// The station's data folder is an absolute path the medium creates on its first
// request (the press uses C:\ProgramData\Fraktal\PressDemo\).
METHOD A_file_medium_creates_its_folder
TEST('A_file_medium_creates_its_folder');
_t4(IN := _s4 < 99, PT := TEST_TIMEOUT);
IF _t4.Q AND (_s4 < 99) THEN
    AssertTrue(Condition := FALSE, Message := CONCAT('timed out in step ', INT_TO_STRING(_s4)));
    _s4 := 99;
    TEST_FINISHED();
    RETURN;
END_IF
_f4.Cyclic();
CASE _s4 OF
    0:
        AssertTrue(Condition := _m4.Setup(Folder := GENERIC_FOLDER, Where := Tc2_System.PATH_GENERIC),
            Message := 'an absolute folder is accepted');
        _k4 := _m4.M_StartWrite(Key := _M_Key(Name := 'Folder'), pData := ADR(_docA),
            Size := SIZEOF(_docA));
        _s4 := 1;
    1:
        IF _m4.M_Poll(Ticket := _k4, Result := _r4) THEN
            AssertTrue(Condition := _r4.Ok, Message := 'the document is written into the folder');
            _k4 := _m4.M_StartRead(Key := _M_Key(Name := 'Folder'), pData := ADR(_buf),
                Size := SIZEOF(_buf));
            _s4 := 2;
        END_IF
    2:
        IF _m4.M_Poll(Ticket := _k4, Result := _r4) THEN
            AssertTrue(Condition := _r4.Found AND (_r4.Length = SIZEOF(_docA)),
                Message := 'and read back from it');
            _f4.M_Delete(Path := CONCAT(GENERIC_FOLDER, CONCAT(_M_Key(Name := 'Folder'), '.a')),
                Where := Tc2_System.PATH_GENERIC);
            _s4 := 3;
        END_IF
    3:
        IF NOT _f4.Busy THEN
            AssertFalse(Condition := _f4.Error, Message := 'the file was where the medium said');
            _s4 := 99;
            TEST_FINISHED();
        END_IF
    99:
        ;
ELSE
    _s4 := 99;
END_CASE
END_METHOD

// Regression (live acceptance 2026-10-06): with the newest copy in slot a and an
// older one in slot b, a fresh run returned nothing - the payload check compared
// slot a against slot b's header - and its next write then replaced slot a, the
// newest copy. A fresh medium must read slot a, and must write the next copy to b.
METHOD The_newest_copy_wins_in_either_slot
VAR
    key : STRING(80);
END_VAR
TEST('The_newest_copy_wins_in_either_slot');
_t5(IN := _s5 < 99, PT := TEST_TIMEOUT);
IF _t5.Q AND (_s5 < 99) THEN
    AssertTrue(Condition := FALSE, Message := CONCAT('timed out in step ', INT_TO_STRING(_s5)));
    _s5 := 99;
    TEST_FINISHED();
    RETURN;
END_IF
key := _M_Key(Name := 'Slots');
_f5.Cyclic();
CASE _s5 OF
    0:      // generation 1 -> a, 2 -> b, 3 -> a
        _m5.Setup(Folder := '', Where := Tc2_System.PATH_BOOTPATH);
        _k5 := _m5.M_StartWrite(Key := key, pData := ADR(_docA), Size := SIZEOF(_docA));
        _s5 := 1;
    1:
        IF _m5.M_Poll(Ticket := _k5, Result := _r5) THEN
            _k5 := _m5.M_StartWrite(Key := key, pData := ADR(_docB), Size := SIZEOF(_docB));
            _s5 := 2;
        END_IF
    2:
        IF _m5.M_Poll(Ticket := _k5, Result := _r5) THEN
            _k5 := _m5.M_StartWrite(Key := key, pData := ADR(_docA), Size := SIZEOF(_docA));
            _s5 := 3;
        END_IF
    3:
        IF _m5.M_Poll(Ticket := _k5, Result := _r5) THEN
            AssertTrue(Condition := _r5.Ok, Message := 'three copies written');
            _m6.Setup(Folder := '', Where := Tc2_System.PATH_BOOTPATH);
            MEMSET(destAddr := ADR(_buf), fillByte := 0, n := SIZEOF(_buf));
            _k5 := _m6.M_StartRead(Key := key, pData := ADR(_buf), Size := SIZEOF(_buf));
            _s5 := 4;
        END_IF
    4:      // a fresh run reads the newest copy, which is in slot a
        IF _m6.M_Poll(Ticket := _k5, Result := _r5) THEN
            AssertTrue(Condition := _r5.Ok AND _r5.Found AND NOT _r5.Lost,
                Message := 'a fresh run finds the newest copy in slot a');
            AssertEquals_UDINT(Expected := SIZEOF(_docA), Actual := _r5.Length,
                Message := 'generation 3, not the older copy in slot b');
            _k5 := _m6.M_StartWrite(Key := key, pData := ADR(_docB), Size := SIZEOF(_docB));
            _s5 := 5;
        END_IF
    5:
        IF _m6.M_Poll(Ticket := _k5, Result := _r5) THEN
            AssertTrue(Condition := _r5.Ok, Message := 'generation 4 is written');
            // It must have replaced slot b: remove b and slot a still holds generation 3.
            _f5.M_Delete(Path := CONCAT(key, '.b'), Where := Tc2_System.PATH_BOOTPATH);
            _s5 := 6;
        END_IF
    6:
        IF NOT _f5.Busy THEN
            _m7.Setup(Folder := '', Where := Tc2_System.PATH_BOOTPATH);
            _k5 := _m7.M_StartRead(Key := key, pData := ADR(_buf), Size := SIZEOF(_buf));
            _s5 := 7;
        END_IF
    7:
        IF _m7.M_Poll(Ticket := _k5, Result := _r5) THEN
            AssertTrue(Condition := _r5.Found, Message := 'slot a was not overwritten');
            AssertEquals_UDINT(Expected := SIZEOF(_docA), Actual := _r5.Length,
                Message := 'the next write went to the slot without the newest copy');
            _f5.M_Delete(Path := CONCAT(key, '.a'), Where := Tc2_System.PATH_BOOTPATH);
            _s5 := 8;
        END_IF
    8:
        IF NOT _f5.Busy THEN
            _s5 := 99;
            TEST_FINISHED();
        END_IF
    99:
        ;
ELSE
    _s5 := 99;
END_CASE
END_METHOD

END_FUNCTION_BLOCK

// ---- Fraktal_Tests/FB_LiveConfig_Tests.TcPOU
// Core §3.8b under test: a root's live configuration and its parameter sets on a
// persistence medium, through the surface a station uses - SetPersistMedium and
// SetConfigStore - and the real file service of the test runtime.
//
// A "restart" is a second root instance with the same identity over the same
// files. Each test uses per-run names and removes what it wrote.
FUNCTION_BLOCK FB_LiveConfig_Tests EXTENDS TcUnit.FB_TestSuite
VAR
    _tag     : STRING(24);
    _name    : STRING(80);
    _garbage : ARRAY[0..15] OF BYTE := [16(16#5A)];
    _report  : ST_ReleaseReport;
    _s1 : INT;
    _t1 : TON;
    _m1 : FB_FilePersistMedium;
    _m2 : FB_FilePersistMedium;
    _r1 : FB_LocalRecipeProvider;
    _r2 : FB_LocalRecipeProvider;
    _rec0a, _recAa, _recBa : ST_ProbeModelParCfg;
    _rec0b, _recAb, _recBb : ST_ProbeModelParCfg;
    _u1 : FB_ProbeModelUnit;
    _u2 : FB_ProbeModelUnit;
    _u3 : FB_ProbeModelUnit;
    _f1 : FB_ProbeFileOps;
    _n1 : INT;
    _s2 : INT;
    _t2 : TON;
    _m3  : FB_FilePersistMedium;
    _m3b : FB_FilePersistMedium;
    _st1 : FB_MediumConfigStore;
    _st2 : FB_MediumConfigStore;
    _st3 : FB_MediumConfigStore;
    _f2 : FB_ProbeFileOps;
    _s3 : INT;
    _t3 : TON;
    _m4 : FB_FilePersistMedium;
    _st4 : FB_MediumConfigStore;
    _r4 : FB_LocalRecipeProvider;
    _rec4 : ST_ProbeModelParCfg;
    _u4 : FB_ProbeModelUnit;
    _f3 : FB_ProbeFileOps;
END_VAR
VAR CONSTANT
    TEST_TIMEOUT : TIME := T#60S;
END_VAR

IF _tag = '' THEN
    _tag := ULINT_TO_STRING(Tc2_Utilities.F_GetSystemTime() MOD 1000000000000);
    _name := CONCAT('Live', _tag);
END_IF
Station_and_model_data_come_back_from_their_documents();
Parameter_sets_come_back_from_the_medium();
A_saved_set_is_pending_until_its_document_is_written();

// Start names the restore while the documents are being read back.
METHOD PRIVATE _M_Restoring : BOOL
VAR_IN_OUT
    Unit : FB_ProbeModelUnit;
END_VAR
VAR
    i : INT;
END_VAR
_M_Restoring := FALSE;
Unit.ReleaseReportStart(Report := _report);
FOR i := 1 TO MIN(_report.Count, PL_Fraktal.MAX_RELEASE_REASONS) DO
    IF _report.Reasons[i].Description = 'std.release.configRestoring' THEN
        _M_Restoring := TRUE;
    END_IF
END_FOR
END_METHOD

// The n-th file of this root's live documents: station, then models 1 and 2,
// each slot a then b.
METHOD PRIVATE _M_LiveFile : STRING(255)
VAR_INPUT
    Index : INT;
END_VAR
VAR
    doc : STRING(40);
END_VAR
CASE Index / 2 OF
    0: doc := '.station';
    1: doc := '.model1';
ELSE
    doc := '.model2';
END_CASE
IF (Index MOD 2) = 0 THEN
    _M_LiveFile := CONCAT(_name, CONCAT(doc, '.a'));
ELSE
    _M_LiveFile := CONCAT(_name, CONCAT(doc, '.b'));
END_IF
END_METHOD

METHOD Station_and_model_data_come_back_from_their_documents
TEST('Station_and_model_data_come_back_from_their_documents');
_t1(IN := _s1 < 99, PT := TEST_TIMEOUT);
IF _t1.Q AND (_s1 < 99) THEN
    AssertTrue(Condition := FALSE, Message := CONCAT('timed out in step ', INT_TO_STRING(_s1)));
    _s1 := 99;
    TEST_FINISHED();
    RETURN;
END_IF
_f1.Cyclic();
CASE _s1 OF
    0:      // first run
        _rec0a.Speed := 1;
        _recAa.Speed := 10;
        _recBa.Speed := 20;
        _r1.Register(ModelCode := '', RecipeKey := 'ProbeModel', pData := ADR(_rec0a), Size := SIZEOF(_rec0a));
        _r1.Register(ModelCode := 'A', RecipeKey := 'ProbeModel', pData := ADR(_recAa), Size := SIZEOF(_recAa));
        _r1.Register(ModelCode := 'B', RecipeKey := 'ProbeModel', pData := ADR(_recBa), Size := SIZEOF(_recBa));
        _u1.ParCfg := _rec0a;
        _u1.Setup(Name := _name, Provider := _r1);
        _m1.Setup(Folder := '', Where := Tc2_System.PATH_BOOTPATH);
        AssertTrue(Condition := _u1.SetPersistMedium(Medium := _m1), Message := 'the medium is accepted');
        _u1();
        AssertFalse(Condition := _u1.WriteConfig(TargetPath := _name, WriteKey := 'probe.limit',
            Revision := 1, TextValue := '42'),
            Message := 'a write before the documents are back is refused: the restore would replay over it');
        AssertTrue(Condition := _M_Restoring(Unit := _u1), Message := 'and Start names the restore');
        _s1 := 1;
    1:
        _u1();
        IF NOT _M_Restoring(Unit := _u1) THEN
            AssertFalse(Condition := _u1.ConfigPersist.RestoreLost,
                Message := 'documents that never existed lost nothing');
            AssertTrue(Condition := _u1.WriteConfig(TargetPath := _name, WriteKey := 'probe.limit',
                Revision := 1, TextValue := '42'), Message := 'a station value is written');
            AssertTrue(Condition := _u1.WriteModelConfig(ModelIndex := 2, TargetPath := _name,
                WriteKey := 'probe.speed', Revision := 1, TextValue := '25'),
                Message := 'a model value of model B is written');
            AssertTrue(Condition := _u1.ConfigPersist.Pending, Message := 'live, not yet durable');
            _s1 := 2;
        END_IF
    2:
        _u1();
        IF NOT _u1.ConfigPersist.Pending THEN
            AssertFalse(Condition := _u1.ConfigPersist.Failed,
                Message := 'the documents are written within the declared window');
            _s1 := 3;
        END_IF
    3:      // restart: a new instance of the same root over the same files
        _rec0b.Speed := 1;
        _recAb.Speed := 10;
        _recBb.Speed := 20;
        _r2.Register(ModelCode := '', RecipeKey := 'ProbeModel', pData := ADR(_rec0b), Size := SIZEOF(_rec0b));
        _r2.Register(ModelCode := 'A', RecipeKey := 'ProbeModel', pData := ADR(_recAb), Size := SIZEOF(_recAb));
        _r2.Register(ModelCode := 'B', RecipeKey := 'ProbeModel', pData := ADR(_recBb), Size := SIZEOF(_recBb));
        _u2.ParCfg := _rec0b;
        _u2.Setup(Name := _name, Provider := _r2);
        _m2.Setup(Folder := '', Where := Tc2_System.PATH_BOOTPATH);
        _u2.SetPersistMedium(Medium := _m2);
        _u2();
        _s1 := 4;
    4:
        _u2();
        IF NOT _M_Restoring(Unit := _u2) THEN
            AssertEquals_DINT(Expected := 42, Actual := _u2.StationLimit,
                Message := 'the station value comes back from its document');
            AssertEquals_DINT(Expected := 25, Actual := _recBb.Speed,
                Message := 'model B$'s value comes back into B$'s record');
            AssertEquals_DINT(Expected := 10, Actual := _recAb.Speed,
                Message := 'model A keeps its own value');
            AssertFalse(Condition := _u2.ConfigPersist.RestoreLost, Message := 'nothing was lost');
            _s1 := 5;
        END_IF
    5:      // damage both copies of the station document
        _u2();
        IF NOT _u2.ConfigPersist.Pending AND _f1.M_Write(Path := _M_LiveFile(Index := 0),
                Where := Tc2_System.PATH_BOOTPATH, pData := ADR(_garbage), Size := SIZEOF(_garbage)) THEN
            _s1 := 6;
        END_IF
    6:
        IF NOT _f1.Busy AND _f1.M_Write(Path := _M_LiveFile(Index := 1),
                Where := Tc2_System.PATH_BOOTPATH, pData := ADR(_garbage), Size := SIZEOF(_garbage)) THEN
            _s1 := 7;
        END_IF
    7:      // restart over the medium that confirmed the writes
        IF NOT _f1.Busy THEN
            _u3.ParCfg := _rec0b;
            _u3.Setup(Name := _name, Provider := _r2);
            _u3.SetPersistMedium(Medium := _m2);
            _u3();
            _s1 := 8;
        END_IF
    8:
        _u3();
        IF NOT _M_Restoring(Unit := _u3) THEN
            _u3();                      // the loss is drained on the next scan
            AssertTrue(Condition := _u3.ConfigPersist.RestoreLost,
                Message := 'a station document confirmed and then lost is a loss (3.8b)');
            AssertEquals_STRING(Expected := CONCAT(_name, '.station'),
                Actual := _u3.ConfigPersist.LostPath, Message := 'named by its document');
            AssertTrue(Condition := F_ProbeAlarmActive(pLog := ADR(_u3.AlarmLog),
                Reason := E_Reason.CONFIG_RESTORE_LOST, Source := CONCAT(_name, '.station')),
                Message := 'and announced');
            AssertEquals_DINT(Expected := 5, Actual := _u3.StationLimit,
                Message := 'nothing is taken from a damaged document');
            AssertEquals_DINT(Expected := 25, Actual := _recBb.Speed,
                Message := 'an intact model document still restores');
            _s1 := 9;
        END_IF
    9:      // the baseline is rewritten; then remove every file
        _u3();
        IF NOT _u3.ConfigPersist.Pending THEN
            _n1 := 0;
            _s1 := 10;
        END_IF
    10:
        IF _n1 > 5 THEN
            _s1 := 99;
            TEST_FINISHED();
        ELSIF NOT _f1.Busy AND _f1.M_Delete(Path := _M_LiveFile(Index := _n1),
                Where := Tc2_System.PATH_BOOTPATH) THEN
            _n1 := _n1 + 1;
        END_IF
    99:
        ;
ELSE
    _s1 := 99;
END_CASE
END_METHOD

METHOD Parameter_sets_come_back_from_the_medium
VAR
    info   : ST_ConfigSetInfo;
    record : ST_ConfigRecord;
    prefix : STRING(60);
END_VAR
TEST('Parameter_sets_come_back_from_the_medium');
_t2(IN := _s2 < 99, PT := TEST_TIMEOUT);
IF _t2.Q AND (_s2 < 99) THEN
    AssertTrue(Condition := FALSE, Message := CONCAT('timed out in step ', INT_TO_STRING(_s2)));
    _s2 := 99;
    TEST_FINISHED();
    RETURN;
END_IF
prefix := CONCAT('FrkSets_', _tag);
_f2.Cyclic();
CASE _s2 OF
    0:
        _m3.Setup(Folder := '', Where := Tc2_System.PATH_BOOTPATH);
        AssertTrue(Condition := _st1.Setup(Medium := _m3, KeyPrefix := prefix),
            Message := 'the store takes the medium');
        info.SetName := 'Recipe';
        info.RootIdentity := 'Test.Sets';
        info.SetSchema := 1;
        info.ConfigRev := 7;
        info.Kind := E_ConfigKind.STATION_CFG;
        AssertFalse(Condition := _st1.M_SaveBegin(Info := info),
            Message := 'no save before the stored sets are back');
        _s2 := 1;
    1:
        _st1.M_Cyclic();
        IF _st1.Restored THEN
            AssertEquals_INT(Expected := 0, Actual := _st1.M_Count(), Message := 'an empty medium');
            AssertFalse(Condition := _st1.RestoreLost, Message := 'lost nothing');
            info.SetName := 'Recipe';
            info.RootIdentity := 'Test.Sets';
            info.SetSchema := 1;
            info.ConfigRev := 7;
            info.Kind := E_ConfigKind.STATION_CFG;
            AssertTrue(Condition := _st1.M_SaveBegin(Info := info), Message := 'a save opens');
            record.Scope := 'Test.Sets';
            record.WriteKey := 'probe.limit';
            record.Revision := 1;
            record.Kind := E_ConfigKind.STATION_CFG;
            record.ValueType := E_ConfigValueType.NUMBER;
            record.ValueText := '42';
            _st1.M_SaveRecord(Record := record);
            record.WriteKey := 'probe.text';
            record.ValueType := E_ConfigValueType.TEXT;
            record.ValueText := 'with "quotes", a \ and a , comma';
            _st1.M_SaveRecord(Record := record);
            AssertTrue(Condition := _st1.M_SaveCommit(), Message := 'and commits');
            AssertFalse(Condition := _st1.Durable, Message := 'live, not yet written');
            _s2 := 2;
        END_IF
    2:
        _st1.M_Cyclic();
        IF _st1.Durable THEN
            _m3b.Setup(Folder := '', Where := Tc2_System.PATH_BOOTPATH);
            _st2.Setup(Medium := _m3b, KeyPrefix := prefix);
            _s2 := 3;
        END_IF
    3:
        _st2.M_Cyclic();
        IF _st2.Restored THEN
            AssertEquals_INT(Expected := 1, Actual := _st2.M_Count(), Message := 'the set comes back');
            AssertTrue(Condition := _st2.M_ReadInfo(SetName := 'Recipe', Info := info),
                Message := 'under its name');
            AssertEquals_INT(Expected := 2, Actual := info.RecordCount, Message := 'whole');
            AssertEquals_STRING(Expected := 'Test.Sets', Actual := info.RootIdentity,
                Message := 'with the identity of the root that took it');
            AssertTrue(Condition := _st2.M_ReadRecord(SetName := 'Recipe', Index := 2,
                Record := record), Message := 'a record reads back');
            AssertEquals_STRING(Expected := 'with "quotes", a \ and a , comma',
                Actual := record.ValueText, Message := 'a text value survives the file exactly');
            AssertTrue(Condition := _st2.M_Delete(SetName := 'Recipe'), Message := 'the set is deleted');
            _s2 := 4;
        END_IF
    4:
        _st2.M_Cyclic();
        IF _st2.Durable THEN
            _st3.Setup(Medium := _m3b, KeyPrefix := prefix);
            _s2 := 5;
        END_IF
    5:
        _st3.M_Cyclic();
        IF _st3.Restored THEN
            AssertEquals_INT(Expected := 0, Actual := _st3.M_Count(),
                Message := 'a deleted set stays deleted');
            AssertFalse(Condition := _st3.RestoreLost, Message := 'by intent, not lost');
            _f2.M_Delete(Path := CONCAT(prefix, '.set1.a'), Where := Tc2_System.PATH_BOOTPATH);
            _s2 := 6;
        END_IF
    6:
        IF NOT _f2.Busy THEN
            _f2.M_Delete(Path := CONCAT(prefix, '.set1.b'), Where := Tc2_System.PATH_BOOTPATH);
            _s2 := 7;
        END_IF
    7:
        IF NOT _f2.Busy THEN
            _s2 := 99;
            TEST_FINISHED();
        END_IF
    99:
        ;
ELSE
    _s2 := 99;
END_CASE
END_METHOD

// The root finds the store's own writer (__QUERYINTERFACE) and drives it, so a
// saved set is PersistPending until its document is written - one SetConfigStore.
METHOD A_saved_set_is_pending_until_its_document_is_written
VAR
    prefix : STRING(60);
END_VAR
TEST('A_saved_set_is_pending_until_its_document_is_written');
_t3(IN := _s3 < 99, PT := TEST_TIMEOUT);
IF _t3.Q AND (_s3 < 99) THEN
    AssertTrue(Condition := FALSE, Message := CONCAT('timed out in step ', INT_TO_STRING(_s3)));
    _s3 := 99;
    TEST_FINISHED();
    RETURN;
END_IF
prefix := CONCAT('FrkRootSets_', _tag);
_f3.Cyclic();
CASE _s3 OF
    0:
        _rec4.Speed := 3;
        _r4.Register(ModelCode := '', RecipeKey := 'ProbeModel', pData := ADR(_rec4), Size := SIZEOF(_rec4));
        _u4.ParCfg := _rec4;
        _u4.Setup(Name := CONCAT('Sets', _tag), Provider := _r4);
        _m4.Setup(Folder := '', Where := Tc2_System.PATH_BOOTPATH);
        _st4.Setup(Medium := _m4, KeyPrefix := prefix);
        AssertTrue(Condition := _u4.SetConfigStore(Store := _st4), Message := 'the store is wired');
        _u4();
        _s3 := 1;
    1:
        _u4();                          // the root, not the test, drives the store
        IF _st4.Restored THEN
            AssertEquals_DINT(Expected := TO_DINT(E_ConfigStore.FILE_JSON),
                Actual := TO_DINT(_u4.ConfigPersist.StoreKind), Message := 'published as a file store');
            AssertTrue(Condition := _u4.SaveConfigSet(SetName := 'Commissioned',
                Kind := E_ConfigKind.STATION_CFG), Message := 'a station set is saved');
            AssertTrue(Condition := _u4.ConfigPersist.Pending, Message := 'pending');
            _s3 := 2;
        END_IF
    2:
        _u4();
        IF NOT _u4.ConfigPersist.Pending THEN
            AssertTrue(Condition := _st4.Durable,
                Message := 'Pending cleared only once the set document is written');
            AssertFalse(Condition := _u4.ConfigPersist.Failed, Message := 'without a failure');
            _f3.M_Delete(Path := CONCAT(prefix, '.set1.a'), Where := Tc2_System.PATH_BOOTPATH);
            _s3 := 3;
        END_IF
    3:
        IF NOT _f3.Busy THEN
            _s3 := 99;
            TEST_FINISHED();
        END_IF
    99:
        ;
ELSE
    _s3 := 99;
END_CASE
END_METHOD

END_FUNCTION_BLOCK

// ---- Fraktal_Tests/PRG_PlatformAcceptance.TcPOU
// Live acceptance harness on the ISOLATED test runtime - not a TcUnit suite. After
// the suites finish it keeps running, so an operator can read, over ADS, what the
// real target providers report while they change the target underneath them:
// stop/start the Windows clock observer or Windows Time, corrupt its record, and
// see the Device Manager and EtherCAT master answer (or, on a host without them,
// stay explicitly unavailable). It writes no global: GVL_FraktalTime stays the
// suites' to set. CLOCK_FILE is a dedicated acceptance path, never the
// installed observer's protected default directory.
//
// Retention is wired as the press wires it (§3.8b, IMPLEMENTATION_NOTES §163): one
// file medium in DATA_FOLDER holds the user table (AccessUsers, key
// 'Acceptance.users'), LiveUnit's station and model documents, and LiveSets'
// parameter sets. The same instances, their confirmation markers and their files
// are the only way to accept retention across a real runtime restart or download.
// The acceptance script registers test users by writing RegisterUser/Pin/Level and
// logs in through AccessUnit.Access exactly as an HMI does; it edits LiveUnit's
// values through SetLimit/SetModelSpeed/SaveSet, which call the root's own write
// methods.
PROGRAM PRG_PlatformAcceptance
VAR
    Clock : FB_TcWindowsTime;
    Ipc : FB_TcIpcDiagnostics;
    Bus : FB_EcBusHealth;
    {attribute 'OPC.UA.DA' := '0'}
    _topology : FB_IoTopologyPublisher;
    _setup : BOOL;
    _noMaster : T_AmsNetIdArr;      // all zero: derive the local master's NetId
    AccessUnit : FB_ProbeUnit;
    AccessUsers : FB_LocalAccessProvider;
    RegisterUser : STRING(32);      // written by the acceptance script, consumed here
    RegisterPin : STRING(32);
    RegisterLevel : E_AccessLevel;
    Registered : UDINT;             // accepted registrations this run
    Storage : FB_FilePersistMedium;
    LiveRecipes : FB_LocalRecipeProvider;
    LiveRec0 : ST_ProbeModelParCfg := (Speed := 1);
    LiveRecA : ST_ProbeModelParCfg := (Speed := 10);
    LiveRecB : ST_ProbeModelParCfg := (Speed := 20);
    LiveSets : FB_MediumConfigStore;
    LiveUnit : FB_ProbeModelUnit;
    SetLimit : DINT;                // written by the script: 0 = nothing to do
    SetModelSpeed : DINT;           // model B (AvailableModels[2]); 0 = nothing to do
    SaveSet : BOOL;
    LastWriteOk : BOOL;
    Writes : UDINT;                 // accepted writes this run
    // File commands into DATA_FOLDER through the PLC's own file service (the
    // runtime's account owns the files; an ordinary host user may only read them).
    DamageFile : STRING(80);        // overwritten with 16 bytes of 16#5A
    RemoveFile : STRING(80);        // deleted
    ObstructFile : STRING(80);      // a directory created in its place
    ClearObstruction : STRING(80);  // that directory removed
    FileOps : UDINT;                // completed file commands this run
    FileOpError : UDINT;            // ErrorId of the last one (0 = none)
    {attribute 'OPC.UA.DA' := '0'}
    _files : FB_ProbeFileOps;
    _garbage : ARRAY[0..15] OF BYTE := [16(16#5A)];
    _fileOpBusy : BOOL;
END_VAR
VAR CONSTANT
    CLOCK_FILE : STRING(80) := 'C:\ProgramData\Fraktal\ClockAcceptance\quality.bin';
    DATA_FOLDER : STRING(80) := 'C:\ProgramData\Fraktal\Acceptance\';
END_VAR

IF NOT _setup THEN
    _setup := TRUE;
    // No slave is mapped: only the always-on master sample runs.
    Bus.Setup(Publisher := _topology, MasterNetIdArr := _noMaster,
        FirstSlaveNode := 1, SlaveCount := 0, MasterNodeIndex := 0);
    Storage.Setup(Folder := DATA_FOLDER, Where := Tc2_System.PATH_GENERIC);
    AccessUsers.M_UseMedium(Medium := Storage);
    AccessUsers.M_UseKey(Key := 'Acceptance.users');
    AccessUnit.Setup('Acceptance');
    AccessUnit();
    AccessUnit.Access.Setup(Provider := AccessUsers, pAlarmLog := ADR(AccessUnit.AlarmLog));
    LiveRecipes.Register(ModelCode := '', RecipeKey := 'ProbeModel', pData := ADR(LiveRec0), Size := SIZEOF(LiveRec0));
    LiveRecipes.Register(ModelCode := 'A', RecipeKey := 'ProbeModel', pData := ADR(LiveRecA), Size := SIZEOF(LiveRecA));
    LiveRecipes.Register(ModelCode := 'B', RecipeKey := 'ProbeModel', pData := ADR(LiveRecB), Size := SIZEOF(LiveRecB));
    LiveUnit.ParCfg := LiveRec0;
    LiveUnit.Setup(Name := 'AcceptanceLive', Provider := LiveRecipes);
    LiveSets.Setup(Medium := Storage, KeyPrefix := 'AcceptanceLive.sets');
    LiveUnit.SetConfigStore(Store := LiveSets);
    LiveUnit.SetPersistMedium(Medium := Storage);
END_IF
IF SetLimit <> 0 THEN
    LastWriteOk := LiveUnit.WriteConfig(TargetPath := 'AcceptanceLive', WriteKey := 'probe.limit',
        Revision := 1, TextValue := DINT_TO_STRING(SetLimit));
    SetLimit := 0;
    IF LastWriteOk THEN Writes := Writes + 1; END_IF
END_IF
IF SetModelSpeed <> 0 THEN
    LastWriteOk := LiveUnit.WriteModelConfig(ModelIndex := 2, TargetPath := 'AcceptanceLive',
        WriteKey := 'probe.speed', Revision := 1, TextValue := DINT_TO_STRING(SetModelSpeed));
    SetModelSpeed := 0;
    IF LastWriteOk THEN Writes := Writes + 1; END_IF
END_IF
IF SaveSet THEN
    LastWriteOk := LiveUnit.SaveConfigSet(SetName := 'AcceptanceSet', Kind := E_ConfigKind.STATION_CFG);
    SaveSet := FALSE;
    IF LastWriteOk THEN Writes := Writes + 1; END_IF
END_IF
_files.Cyclic();
IF _fileOpBusy AND NOT _files.Busy THEN
    _fileOpBusy := FALSE;
    FileOps := FileOps + 1;
    FileOpError := _files.ErrorId;
END_IF
IF NOT _files.Busy THEN
    IF DamageFile <> '' THEN
        _fileOpBusy := _files.M_Write(Path := CONCAT(DATA_FOLDER, DamageFile),
            Where := Tc2_System.PATH_GENERIC, pData := ADR(_garbage), Size := SIZEOF(_garbage));
        DamageFile := '';
    ELSIF RemoveFile <> '' THEN
        _fileOpBusy := _files.M_Delete(Path := CONCAT(DATA_FOLDER, RemoveFile),
            Where := Tc2_System.PATH_GENERIC);
        RemoveFile := '';
    ELSIF ObstructFile <> '' THEN
        _fileOpBusy := _files.M_MakeDir(Path := CONCAT(DATA_FOLDER, ObstructFile),
            Where := Tc2_System.PATH_GENERIC);
        ObstructFile := '';
    ELSIF ClearObstruction <> '' THEN
        _fileOpBusy := _files.M_RemoveDir(Path := CONCAT(DATA_FOLDER, ClearObstruction),
            Where := Tc2_System.PATH_GENERIC);
        ClearObstruction := '';
    END_IF
END_IF
LiveUnit();
IF RegisterUser <> '' THEN
    IF AccessUsers.Register(User := RegisterUser, Pin := RegisterPin, Level := RegisterLevel) THEN
        Registered := Registered + 1;
    END_IF
    RegisterUser := '';
    RegisterPin := '';
END_IF
AccessUnit();
Clock.Cyclic(FilePath := CLOCK_FILE, PollInterval := T#10S, MaximumSampleAge := T#90S,
    MaximumSyncAgeSeconds := 7200, MaximumOffsetUs := 1000);
Ipc.Cyclic();
Bus.M_Refresh();

END_PROGRAM

// ---- Fraktal_Tests/FB_Separator_Tests.TcPOU
// Annex A separator/stopper. T1/T4 are proven once in FB_Base_Tests for every
// inheriting type and are deliberately NOT repeated here (Core S5.7).
//
// The first test is the one that matters most: this type declares NO interlocks
// of its own (S7.2.1), so the suite proves both halves of that contract - nothing
// gates a station that declares nothing, and a condition the application declares
// is fail-closed until the application drives it.
FUNCTION_BLOCK FB_Separator_Tests EXTENDS TcUnit.FB_TestSuite
VAR
    _hal : ST_SeparatorHal;
    _sep : FB_SeparatorCM;
    _halT3 : ST_SeparatorHal;
    _sepT3 : FB_SeparatorCM;
    _halSep : ST_SeparatorHal;
    _sepSep : FB_SeparatorCM;
    _halNo : ST_SeparatorHal;
    _sepNo : FB_SeparatorCM;
    _halOc : ST_SeparatorHal;
    _sepOc : FB_SeparatorCM;
    _halBad : ST_SeparatorHal;
    _sepBad : FB_SeparatorCM;
    _i : INT;
    _w1, _w2, _w3, _w4, _w5, _w6 : BOOL;
END_VAR

Library_declares_no_interlocks_and_application_conditions_are_fail_closed();
Interlock_withholds_the_valve_and_holds_rather_than_faults();
Separate_releases_one_carrier_and_completes();
No_carrier_at_the_separator_faults_10001();
Open_close_confirms_feedback_only_when_configured();
Unsupported_command_is_rejected();

METHOD Library_declares_no_interlocks_and_application_conditions_are_fail_closed
TEST('Library_declares_no_interlocks_and_application_conditions_are_fail_closed');
IF NOT _w1 THEN
    _sep.Setup(Name := 'Sep1', HalRef := _hal, Recipe := 0);
    _sep();
    // S7.2.1: a reusable type publishes no condition it cannot derive. A station
    // that declares nothing is therefore not gated by anything.
    AssertTrue(Condition := _sep.Intlk.AllOk,
        Message := 'a library type that declares no interlock does not gate the station');
    AssertTrue(Condition := _sep.DeclareCondition(Index := 1,
            DescriptionKey := 'std.interlock.areaSafe',
            Reason := E_Reason.INTERLOCK_DROPPED, Bypassable := FALSE),
        Message := 'the application may claim any index');
    _sep();
    // Declaring states an intent to gate, so the fail-closed default holds until
    // the application actually drives it.
    AssertFalse(Condition := _sep.Intlk.AllOk,
        Message := 'a declared but undriven condition is fail-closed');
    AssertTrue(Condition := _sep.SetCondition(Index := 1, Ok := TRUE),
        Message := 'the application drives its own condition');
    _sep();
    AssertTrue(Condition := _sep.Intlk.AllOk,
        Message := 'and the gate clears once it is satisfied');
    AssertFalse(Condition := _sep.DeclareCondition(Index := 0,
            DescriptionKey := 'std.interlock.areaSafe',
            Reason := E_Reason.INTERLOCK_DROPPED, Bypassable := FALSE),
        Message := 'an out-of-range index is refused, not silently ignored');
    _w1 := TRUE;
END_IF
TEST_FINISHED();
END_METHOD

METHOD Interlock_withholds_the_valve_and_holds_rather_than_faults
TEST('Interlock_withholds_the_valve_and_holds_rather_than_faults');
IF NOT _w2 THEN
    _sepT3.Setup(Name := 'SepT3', HalRef := _halT3, Recipe := 0);
    _sepT3.DeclareCondition(Index := 1, DescriptionKey := 'std.interlock.areaSafe',
        Reason := E_Reason.INTERLOCK_DROPPED, Bypassable := FALSE);
    _sepT3.SetCondition(Index := 1, Ok := FALSE);
    _halT3.CarrierAt := TRUE;
    _sepT3.Command := E_SeparatorCommand.SEPARATE;
    _sepT3.Execute := TRUE;
    FOR _i := 1 TO 5 DO
        _sepT3();
    END_FOR
    // T3: the interlock withholds the output, and does so as a HELD wait rather
    // than a fault - losing a condition mid-action is expected, not a defect.
    AssertFalse(Condition := _halT3.ValveOpen,
        Message := 'the valve is withheld while the condition is unsatisfied');
    AssertTrue(Condition := _sepT3.Held, Message := 'and the module reports HELD');
    AssertFalse(Condition := _sepT3.Error, Message := 'not an error');
    AssertEquals_STRING(Expected := 'SepT3', Actual := _sepT3.Status.Diagnostic.SourcePath,
        Message := 'the owning module sets the diagnostic source path');
    _w2 := TRUE;
END_IF
TEST_FINISHED();
END_METHOD

METHOD Separate_releases_one_carrier_and_completes
TEST('Separate_releases_one_carrier_and_completes');
IF NOT _w3 THEN
    _sepSep.Setup(Name := 'SepOk', HalRef := _halSep, Recipe := 0);
    _sepSep.ParCfg.CheckAfter := FALSE;          // stopper variant: no downstream sensor
    _halSep.CarrierAt := TRUE;
    _sepSep.Command := E_SeparatorCommand.SEPARATE;
    _sepSep.Execute := TRUE;
    _sepSep(); _sepSep();
    AssertTrue(Condition := _halSep.ValveOpen, Message := 'opening drives the valve');
    _halSep.CarrierAt := FALSE;                  // the carrier leaves the separator
    _sepSep(); _sepSep(); _sepSep();
    AssertTrue(Condition := _sepSep.Done, Message := 'the command completes');
    AssertTrue(Condition := _sepSep.OutCmd.SeparateOk, Message := 'and reports the release');
    AssertFalse(Condition := _halSep.ValveOpen, Message := 'with the valve closed again');
    _w3 := TRUE;
END_IF
TEST_FINISHED();
END_METHOD

METHOD No_carrier_at_the_separator_faults_10001
TEST('No_carrier_at_the_separator_faults_10001');
IF NOT _w4 THEN
    _sepNo.Setup(Name := 'SepNo', HalRef := _halNo, Recipe := 0);
    // T#0S is the deterministic-timeout idiom used by the sibling suites: a TON
    // with PT := T#0S expires on the call that starts it, so the expiry does not
    // depend on task time elapsing. Calling the FB N times inside one test scan
    // does NOT advance a TON, which is why a small non-zero PT never fires here.
    _sepNo.ParCfg.MaxOpenTime := T#0S;
    _halNo.CarrierAt := FALSE;                   // nothing ever arrives
    _sepNo.Command := E_SeparatorCommand.SEPARATE;
    _sepNo.Execute := TRUE;
    _sepNo(); _sepNo(); _sepNo();
    // T2: the first-out reason is the specific one, not a generic timeout.
    AssertTrue(Condition := _sepNo.Error, Message := 'the command faults');
    AssertEquals_DWORD(Expected := TO_DWORD(PL_ModuleReasons.SEP_NO_CARRIER_AT),
        Actual := _sepNo.ErrorID,
        Message := 'with SEP_NO_CARRIER_AT, not a generic timeout');
    AssertEquals_STRING(Expected := 'SepNo', Actual := _sepNo.Status.Diagnostic.SourcePath,
        Message := 'and the module as its source path');
    AssertFalse(Condition := _halNo.ValveOpen, Message := 'the valve is dropped on fault');
    _w4 := TRUE;
END_IF
TEST_FINISHED();
END_METHOD

METHOD Open_close_confirms_feedback_only_when_configured
TEST('Open_close_confirms_feedback_only_when_configured');
IF NOT _w5 THEN
    _sepOc.Setup(Name := 'SepOc', HalRef := _halOc, Recipe := 0);
    _sepOc.ParCfg.UsesOpenFb := FALSE;           // no feedback wired at this station
    _sepOc.ParCmd.OpenStopper := TRUE;
    _sepOc.Command := E_SeparatorCommand.OPEN_CLOSE;
    _sepOc.Execute := TRUE;
    _sepOc(); _sepOc();
    AssertTrue(Condition := _halOc.ValveOpen, Message := 'the stopper opens');
    AssertTrue(Condition := _sepOc.Done,
        Message := 'and completes without feedback when none is configured');
    _sepOc.Execute := FALSE;
    _sepOc();
    _sepOc.ParCmd.OpenStopper := FALSE;
    _sepOc.Execute := TRUE;
    _sepOc(); _sepOc();
    AssertFalse(Condition := _halOc.ValveOpen, Message := 'closing is immediate');
    AssertTrue(Condition := _sepOc.Done, Message := 'and completes');
    _w5 := TRUE;
END_IF
TEST_FINISHED();
END_METHOD

METHOD Unsupported_command_is_rejected
TEST('Unsupported_command_is_rejected');
IF NOT _w6 THEN
    _sepBad.Setup(Name := 'SepBad', HalRef := _halBad, Recipe := 0);
    _sepBad.Command := E_SeparatorCommand.NONE;   // never a valid request (S5.6)
    _sepBad.Execute := TRUE;
    _sepBad(); _sepBad();
    AssertTrue(Condition := _sepBad.Error, Message := 'an unset command is refused');
    AssertEquals_DWORD(Expected := TO_DWORD(E_Reason.UNSUPPORTED_COMMAND),
        Actual := _sepBad.ErrorID, Message := 'with UNSUPPORTED_COMMAND');
    _w6 := TRUE;
END_IF
TEST_FINISHED();
END_METHOD

END_FUNCTION_BLOCK

// ---- Fraktal_Tests/FB_Engineering_Tests.TcPOU
// Core §7.5 under test: the gate register is write-once and build-driven, the
// standing §7.5.2 annunciation is LOW/SYSTEM/AUTO_RESET, no operator action
// closes it, and §10.5.1 forcing is refused unless the register arms it.
//
// The assertions about OUTPUT_FORCING are written against
// PL_FraktalEngineering.OUTPUT_FORCING rather than against TRUE or FALSE, so the
// suite is green in BOTH images and proves the two are actually coupled - a test
// hard-coded to the production value would pass while the commissioning build
// silently armed nothing.
FUNCTION_BLOCK FB_Engineering_Tests EXTENDS TcUnit.FB_TestSuite
VAR
    _mode : FB_EngineeringMode;
    _overflow : FB_EngineeringMode;
    _u : FB_ProbeUnit;
    _gateMode : FB_EngineeringMode;
    _i : INT;
    _slot : INT;
    _second : INT;
    _w1, _w2, _w3, _w4 : BOOL;
END_VAR

Inactive_gate_is_not_registered_and_declaring_is_idempotent();
Register_overflow_is_reported_not_silent();
Forcing_is_armed_only_by_the_build_constant();
Active_gate_annunciates_low_system_and_no_reset_closes_it();

METHOD Inactive_gate_is_not_registered_and_declaring_is_idempotent
TEST('Inactive_gate_is_not_registered_and_declaring_is_idempotent');
IF NOT _w1 THEN
    // §7.5.1: an inactive gate registers NOTHING - that is what makes a
    // production station's register empty and its gated surfaces invisible
    // rather than merely disabled.
    AssertEquals_INT(Expected := 0,
        Actual := _mode.M_Declare(Name := 'USE_SIMULATION',
            DescriptionKey := 'std.engineering.simulation', Active := FALSE),
        Message := 'an inactive gate is not registered');
    AssertEquals_INT(Expected := 0, Actual := _mode.Count,
        Message := 'so the register stays empty');
    _slot := _mode.M_Declare(Name := 'USE_SIMULATION',
        DescriptionKey := 'std.engineering.simulation', Active := TRUE);
    AssertTrue(Condition := _slot > 0, Message := 'an active gate is registered');
    AssertEquals_STRING(Expected := 'std.engineering.simulation',
        Actual := _mode.Gates[_slot].DescriptionKey,
        Message := 'with the key the standing annunciation will carry');
    // Re-declaring keeps the slot: two callers naming one departure must not
    // produce two standing annunciations for it.
    _second := _mode.M_Declare(Name := 'USE_SIMULATION',
        DescriptionKey := 'std.engineering.simulation', Active := TRUE);
    AssertEquals_INT(Expected := _slot, Actual := _second,
        Message := 'declaring the same gate again keeps its slot');
    AssertEquals_INT(Expected := 1, Actual := _mode.Count,
        Message := 'and does not grow the register');
    AssertFalse(Condition := _mode.Truncated, Message := 'nothing was dropped');
    _w1 := TRUE;
END_IF
TEST_FINISHED();
END_METHOD

METHOD Register_overflow_is_reported_not_silent
VAR
    gateName : STRING(80);
END_VAR
TEST('Register_overflow_is_reported_not_silent');
IF NOT _w2 THEN
    FOR _i := 1 TO PL_Fraktal.MAX_ENGINEERING_GATES + 1 DO
        gateName := CONCAT('GATE_', INT_TO_STRING(_i));
        _overflow.M_Declare(Name := gateName,
            DescriptionKey := 'std.engineering.simulation', Active := TRUE);
    END_FOR
    AssertEquals_INT(Expected := PL_Fraktal.MAX_ENGINEERING_GATES,
        Actual := _overflow.Count, Message := 'the table is bounded (O10)');
    // A gate that overflowed the table would otherwise be a departure nobody is
    // told about - the exact failure §7.5.2 exists to prevent (§5.6).
    AssertTrue(Condition := _overflow.Truncated,
        Message := 'and says so instead of dropping a gate silently');
    _w2 := TRUE;
END_IF
TEST_FINISHED();
END_METHOD

METHOD Forcing_is_armed_only_by_the_build_constant
TEST('Forcing_is_armed_only_by_the_build_constant');
IF NOT _w3 THEN
    // Before anything wires the register, forcing is refused: an unwired Unit is
    // a production Unit (§10.5.1 rule 1, fail closed).
    AssertFalse(Condition := _u.M_ForcePermitted(),
        Message := 'no register wired, so no forcing');
    AssertFalse(Condition := _u.ForceChannel(ChannelPath := 'Test.IO.X',
        Force := TRUE, BoolText := 'true', AnalogText := '0'),
        Message := 'and the request is refused before any resolver runs');
    _u.SetEngineeringMode(Mode := _gateMode);
    AssertTrue(Condition := (_gateMode.ForcingActive = PL_FraktalEngineering.OUTPUT_FORCING),
        Message := 'wiring the register arms forcing iff the build constant says so');
    AssertTrue(Condition := ((_gateMode.Count > 0) = PL_FraktalEngineering.OUTPUT_FORCING),
        Message := 'and an armed force surface always brings its gate with it');
    _w3 := TRUE;
END_IF
TEST_FINISHED();
END_METHOD

METHOD Active_gate_annunciates_low_system_and_no_reset_closes_it
TEST('Active_gate_annunciates_low_system_and_no_reset_closes_it');
IF NOT _w4 THEN
    AssertTrue(Condition := _u.Setup(Name := 'Test.GateUnit'), Message := 'unit sets up');
    _u.SetEngineeringMode(Mode := _gateMode);
    _gateMode.M_Declare(Name := 'USE_SIMULATION',
        DescriptionKey := 'std.engineering.simulation', Active := TRUE);
    _u();
    _slot := _u.AlarmLog.FindActiveSlot(SourcePath := 'Test.GateUnit',
        Description := 'std.engineering.simulation');
    AssertTrue(Condition := _slot > 0, Message := 'the gate is annunciated');
    AssertEquals_DINT(Expected := TO_DINT(E_Severity.LOW),
        Actual := TO_DINT(_u.AlarmLog.Active[_slot].Severity),
        Message := 'at the LOWEST priority (§8.1)');
    AssertEquals_DINT(Expected := TO_DINT(E_Category.SYSTEM),
        Actual := TO_DINT(_u.AlarmLog.Active[_slot].Category),
        Message := 'in the SYSTEM class: this is about the build, not the process');
    AssertEquals_DINT(Expected := TO_DINT(E_ResetClass.AUTO_RESET),
        Actual := TO_DINT(_u.AlarmLog.Active[_slot].ResetClass),
        Message := 'AUTO_RESET, so it never blocks the commissioning it serves');
    AssertFalse(Condition := _u.AlarmLog.Blocking,
        Message := 'and Start stays available');
    // The whole point: no operator action closes this. OperatorReset reaches
    // only MANUAL_RESET events, and the rationalization record is not shelvable.
    _u.AlarmLog.OperatorReset();
    _u();
    AssertTrue(Condition := _u.AlarmLog.FindActiveSlot(SourcePath := 'Test.GateUnit',
        Description := 'std.engineering.simulation') > 0,
        Message := 'an operator reset does not clear it');
    AssertFalse(Condition := _u.AlarmLog.Shelve(Slot := _slot, DurationS := 60),
        Message := 'and shelving cannot silence it either');
    // It is raised ONCE per gate, however long the station runs.
    _u();
    _u();
    AssertEquals_INT(Expected := _gateMode.Count, Actual := _u.AlarmLog.NActive,
        Message := 'one standing event per REGISTERED gate, not one per scan');
    _w4 := TRUE;
END_IF
TEST_FINISHED();
END_METHOD

END_FUNCTION_BLOCK

// ---- Fraktal_Tests/FB_Separator_Tests.TcPOU
// Annex A separator/stopper. T1/T4 are proven once in FB_Base_Tests for every
// inheriting type and are deliberately NOT repeated here (Core S5.7).
//
// The first test is the one that matters most: this type declares NO interlocks
// of its own (S7.2.1), so the suite proves both halves of that contract - nothing
// gates a station that declares nothing, and a condition the application declares
// is fail-closed until the application drives it.
FUNCTION_BLOCK FB_Separator_Tests EXTENDS TcUnit.FB_TestSuite
VAR
    _hal : ST_SeparatorHal;
    _sep : FB_SeparatorCM;
    _halT3 : ST_SeparatorHal;
    _sepT3 : FB_SeparatorCM;
    _halSep : ST_SeparatorHal;
    _sepSep : FB_SeparatorCM;
    _halNo : ST_SeparatorHal;
    _sepNo : FB_SeparatorCM;
    _halOc : ST_SeparatorHal;
    _sepOc : FB_SeparatorCM;
    _halBad : ST_SeparatorHal;
    _sepBad : FB_SeparatorCM;
    _i : INT;
    _w1, _w2, _w3, _w4, _w5, _w6 : BOOL;
END_VAR

Library_declares_no_interlocks_and_application_conditions_are_fail_closed();
Interlock_withholds_the_valve_and_holds_rather_than_faults();
Separate_releases_one_carrier_and_completes();
No_carrier_at_the_separator_faults_10001();
Open_close_confirms_feedback_only_when_configured();
Unsupported_command_is_rejected();

METHOD Library_declares_no_interlocks_and_application_conditions_are_fail_closed
TEST('Library_declares_no_interlocks_and_application_conditions_are_fail_closed');
IF NOT _w1 THEN
    _sep.Setup(Name := 'Sep1', HalRef := _hal, Recipe := 0);
    _sep();
    // S7.2.1: a reusable type publishes no condition it cannot derive. A station
    // that declares nothing is therefore not gated by anything.
    AssertTrue(Condition := _sep.Intlk.AllOk,
        Message := 'a library type that declares no interlock does not gate the station');
    AssertTrue(Condition := _sep.DeclareCondition(Index := 1,
            DescriptionKey := 'std.interlock.areaSafe',
            Reason := E_Reason.INTERLOCK_DROPPED, Bypassable := FALSE),
        Message := 'the application may claim any index');
    _sep();
    // Declaring states an intent to gate, so the fail-closed default holds until
    // the application actually drives it.
    AssertFalse(Condition := _sep.Intlk.AllOk,
        Message := 'a declared but undriven condition is fail-closed');
    AssertTrue(Condition := _sep.SetCondition(Index := 1, Ok := TRUE),
        Message := 'the application drives its own condition');
    _sep();
    AssertTrue(Condition := _sep.Intlk.AllOk,
        Message := 'and the gate clears once it is satisfied');
    AssertFalse(Condition := _sep.DeclareCondition(Index := 0,
            DescriptionKey := 'std.interlock.areaSafe',
            Reason := E_Reason.INTERLOCK_DROPPED, Bypassable := FALSE),
        Message := 'an out-of-range index is refused, not silently ignored');
    _w1 := TRUE;
END_IF
TEST_FINISHED();
END_METHOD

METHOD Interlock_withholds_the_valve_and_holds_rather_than_faults
TEST('Interlock_withholds_the_valve_and_holds_rather_than_faults');
IF NOT _w2 THEN
    _sepT3.Setup(Name := 'SepT3', HalRef := _halT3, Recipe := 0);
    _sepT3.DeclareCondition(Index := 1, DescriptionKey := 'std.interlock.areaSafe',
        Reason := E_Reason.INTERLOCK_DROPPED, Bypassable := FALSE);
    _sepT3.SetCondition(Index := 1, Ok := FALSE);
    _halT3.CarrierAt := TRUE;
    _sepT3.Command := E_SeparatorCommand.SEPARATE;
    _sepT3.Execute := TRUE;
    FOR _i := 1 TO 5 DO
        _sepT3();
    END_FOR
    // T3: the interlock withholds the output, and does so as a HELD wait rather
    // than a fault - losing a condition mid-action is expected, not a defect.
    AssertFalse(Condition := _halT3.ValveOpen,
        Message := 'the valve is withheld while the condition is unsatisfied');
    AssertTrue(Condition := _sepT3.Held, Message := 'and the module reports HELD');
    AssertFalse(Condition := _sepT3.Error, Message := 'not an error');
    AssertEquals_STRING(Expected := 'SepT3', Actual := _sepT3.Status.Diagnostic.SourcePath,
        Message := 'the owning module sets the diagnostic source path');
    _w2 := TRUE;
END_IF
TEST_FINISHED();
END_METHOD

METHOD Separate_releases_one_carrier_and_completes
TEST('Separate_releases_one_carrier_and_completes');
IF NOT _w3 THEN
    _sepSep.Setup(Name := 'SepOk', HalRef := _halSep, Recipe := 0);
    _sepSep.ParCfg.CheckAfter := FALSE;          // stopper variant: no downstream sensor
    _halSep.CarrierAt := TRUE;
    _sepSep.Command := E_SeparatorCommand.SEPARATE;
    _sepSep.Execute := TRUE;
    _sepSep(); _sepSep();
    AssertTrue(Condition := _halSep.ValveOpen, Message := 'opening drives the valve');
    _halSep.CarrierAt := FALSE;                  // the carrier leaves the separator
    _sepSep(); _sepSep(); _sepSep();
    AssertTrue(Condition := _sepSep.Done, Message := 'the command completes');
    AssertTrue(Condition := _sepSep.OutCmd.SeparateOk, Message := 'and reports the release');
    AssertFalse(Condition := _halSep.ValveOpen, Message := 'with the valve closed again');
    _w3 := TRUE;
END_IF
TEST_FINISHED();
END_METHOD

METHOD No_carrier_at_the_separator_faults_10001
TEST('No_carrier_at_the_separator_faults_10001');
IF NOT _w4 THEN
    _sepNo.Setup(Name := 'SepNo', HalRef := _halNo, Recipe := 0);
    // T#0S is the deterministic-timeout idiom used by the sibling suites: a TON
    // with PT := T#0S expires on the call that starts it, so the expiry does not
    // depend on task time elapsing. Calling the FB N times inside one test scan
    // does NOT advance a TON, which is why a small non-zero PT never fires here.
    _sepNo.ParCfg.MaxOpenTime := T#0S;
    _halNo.CarrierAt := FALSE;                   // nothing ever arrives
    _sepNo.Command := E_SeparatorCommand.SEPARATE;
    _sepNo.Execute := TRUE;
    _sepNo(); _sepNo(); _sepNo();
    // T2: the first-out reason is the specific one, not a generic timeout.
    AssertTrue(Condition := _sepNo.Error, Message := 'the command faults');
    AssertEquals_DWORD(Expected := TO_DWORD(PL_ModuleReasons.SEP_NO_CARRIER_AT),
        Actual := _sepNo.ErrorID,
        Message := 'with SEP_NO_CARRIER_AT, not a generic timeout');
    AssertEquals_STRING(Expected := 'SepNo', Actual := _sepNo.Status.Diagnostic.SourcePath,
        Message := 'and the module as its source path');
    AssertFalse(Condition := _halNo.ValveOpen, Message := 'the valve is dropped on fault');
    _w4 := TRUE;
END_IF
TEST_FINISHED();
END_METHOD

METHOD Open_close_confirms_feedback_only_when_configured
TEST('Open_close_confirms_feedback_only_when_configured');
IF NOT _w5 THEN
    _sepOc.Setup(Name := 'SepOc', HalRef := _halOc, Recipe := 0);
    _sepOc.ParCfg.UsesOpenFb := FALSE;           // no feedback wired at this station
    _sepOc.ParCmd.OpenStopper := TRUE;
    _sepOc.Command := E_SeparatorCommand.OPEN_CLOSE;
    _sepOc.Execute := TRUE;
    _sepOc(); _sepOc();
    AssertTrue(Condition := _halOc.ValveOpen, Message := 'the stopper opens');
    AssertTrue(Condition := _sepOc.Done,
        Message := 'and completes without feedback when none is configured');
    _sepOc.Execute := FALSE;
    _sepOc();
    _sepOc.ParCmd.OpenStopper := FALSE;
    _sepOc.Execute := TRUE;
    _sepOc(); _sepOc();
    AssertFalse(Condition := _halOc.ValveOpen, Message := 'closing is immediate');
    AssertTrue(Condition := _sepOc.Done, Message := 'and completes');
    _w5 := TRUE;
END_IF
TEST_FINISHED();
END_METHOD

METHOD Unsupported_command_is_rejected
TEST('Unsupported_command_is_rejected');
IF NOT _w6 THEN
    _sepBad.Setup(Name := 'SepBad', HalRef := _halBad, Recipe := 0);
    _sepBad.Command := E_SeparatorCommand.NONE;   // never a valid request (S5.6)
    _sepBad.Execute := TRUE;
    _sepBad(); _sepBad();
    AssertTrue(Condition := _sepBad.Error, Message := 'an unset command is refused');
    AssertEquals_DWORD(Expected := TO_DWORD(E_Reason.UNSUPPORTED_COMMAND),
        Actual := _sepBad.ErrorID, Message := 'with UNSUPPORTED_COMMAND');
    _w6 := TRUE;
END_IF
TEST_FINISHED();
END_METHOD

END_FUNCTION_BLOCK

// ---- Fraktal_Tests/FB_Engineering_Tests.TcPOU
// Core §7.5 under test: the gate register is write-once and build-driven, the
// standing §7.5.2 annunciation is LOW/SYSTEM/AUTO_RESET, no operator action
// closes it, and §10.5.1 forcing is refused unless the register arms it.
//
// The assertions about OUTPUT_FORCING are written against
// PL_FraktalEngineering.OUTPUT_FORCING rather than against TRUE or FALSE, so the
// suite is green in BOTH images and proves the two are actually coupled - a test
// hard-coded to the production value would pass while the commissioning build
// silently armed nothing.
FUNCTION_BLOCK FB_Engineering_Tests EXTENDS TcUnit.FB_TestSuite
VAR
    _mode : FB_EngineeringMode;
    _overflow : FB_EngineeringMode;
    _u : FB_ProbeUnit;
    _gateMode : FB_EngineeringMode;
    _i : INT;
    _slot : INT;
    _second : INT;
    _w1, _w2, _w3, _w4 : BOOL;
END_VAR

Inactive_gate_is_not_registered_and_declaring_is_idempotent();
Register_overflow_is_reported_not_silent();
Forcing_is_armed_only_by_the_build_constant();
Active_gate_annunciates_low_system_and_no_reset_closes_it();

METHOD Inactive_gate_is_not_registered_and_declaring_is_idempotent
TEST('Inactive_gate_is_not_registered_and_declaring_is_idempotent');
IF NOT _w1 THEN
    // §7.5.1: an inactive gate registers NOTHING - that is what makes a
    // production station's register empty and its gated surfaces invisible
    // rather than merely disabled.
    AssertEquals_INT(Expected := 0,
        Actual := _mode.M_Declare(Name := 'USE_SIMULATION',
            DescriptionKey := 'std.engineering.simulation', Active := FALSE),
        Message := 'an inactive gate is not registered');
    AssertEquals_INT(Expected := 0, Actual := _mode.Count,
        Message := 'so the register stays empty');
    _slot := _mode.M_Declare(Name := 'USE_SIMULATION',
        DescriptionKey := 'std.engineering.simulation', Active := TRUE);
    AssertTrue(Condition := _slot > 0, Message := 'an active gate is registered');
    AssertEquals_STRING(Expected := 'std.engineering.simulation',
        Actual := _mode.Gates[_slot].DescriptionKey,
        Message := 'with the key the standing annunciation will carry');
    // Re-declaring keeps the slot: two callers naming one departure must not
    // produce two standing annunciations for it.
    _second := _mode.M_Declare(Name := 'USE_SIMULATION',
        DescriptionKey := 'std.engineering.simulation', Active := TRUE);
    AssertEquals_INT(Expected := _slot, Actual := _second,
        Message := 'declaring the same gate again keeps its slot');
    AssertEquals_INT(Expected := 1, Actual := _mode.Count,
        Message := 'and does not grow the register');
    AssertFalse(Condition := _mode.Truncated, Message := 'nothing was dropped');
    _w1 := TRUE;
END_IF
TEST_FINISHED();
END_METHOD

METHOD Register_overflow_is_reported_not_silent
VAR
    gateName : STRING(80);
END_VAR
TEST('Register_overflow_is_reported_not_silent');
IF NOT _w2 THEN
    FOR _i := 1 TO PL_Fraktal.MAX_ENGINEERING_GATES + 1 DO
        gateName := CONCAT('GATE_', INT_TO_STRING(_i));
        _overflow.M_Declare(Name := gateName,
            DescriptionKey := 'std.engineering.simulation', Active := TRUE);
    END_FOR
    AssertEquals_INT(Expected := PL_Fraktal.MAX_ENGINEERING_GATES,
        Actual := _overflow.Count, Message := 'the table is bounded (O10)');
    // A gate that overflowed the table would otherwise be a departure nobody is
    // told about - the exact failure §7.5.2 exists to prevent (§5.6).
    AssertTrue(Condition := _overflow.Truncated,
        Message := 'and says so instead of dropping a gate silently');
    _w2 := TRUE;
END_IF
TEST_FINISHED();
END_METHOD

METHOD Forcing_is_armed_only_by_the_build_constant
TEST('Forcing_is_armed_only_by_the_build_constant');
IF NOT _w3 THEN
    // Before anything wires the register, forcing is refused: an unwired Unit is
    // a production Unit (§10.5.1 rule 1, fail closed).
    AssertFalse(Condition := _u.M_ForcePermitted(),
        Message := 'no register wired, so no forcing');
    AssertFalse(Condition := _u.ForceChannel(ChannelPath := 'Test.IO.X',
        Force := TRUE, BoolText := 'true', AnalogText := '0'),
        Message := 'and the request is refused before any resolver runs');
    _u.SetEngineeringMode(Mode := _gateMode);
    AssertTrue(Condition := (_gateMode.ForcingActive = PL_FraktalEngineering.OUTPUT_FORCING),
        Message := 'wiring the register arms forcing iff the build constant says so');
    AssertTrue(Condition := ((_gateMode.Count > 0) = PL_FraktalEngineering.OUTPUT_FORCING),
        Message := 'and an armed force surface always brings its gate with it');
    _w3 := TRUE;
END_IF
TEST_FINISHED();
END_METHOD

METHOD Active_gate_annunciates_low_system_and_no_reset_closes_it
TEST('Active_gate_annunciates_low_system_and_no_reset_closes_it');
IF NOT _w4 THEN
    AssertTrue(Condition := _u.Setup(Name := 'Test.GateUnit'), Message := 'unit sets up');
    _u.SetEngineeringMode(Mode := _gateMode);
    _gateMode.M_Declare(Name := 'USE_SIMULATION',
        DescriptionKey := 'std.engineering.simulation', Active := TRUE);
    _u();
    _slot := _u.AlarmLog.FindActiveSlot(SourcePath := 'Test.GateUnit',
        Description := 'std.engineering.simulation');
    AssertTrue(Condition := _slot > 0, Message := 'the gate is annunciated');
    AssertEquals_DINT(Expected := TO_DINT(E_Severity.LOW),
        Actual := TO_DINT(_u.AlarmLog.Active[_slot].Severity),
        Message := 'at the LOWEST priority (§8.1)');
    AssertEquals_DINT(Expected := TO_DINT(E_Category.SYSTEM),
        Actual := TO_DINT(_u.AlarmLog.Active[_slot].Category),
        Message := 'in the SYSTEM class: this is about the build, not the process');
    AssertEquals_DINT(Expected := TO_DINT(E_ResetClass.AUTO_RESET),
        Actual := TO_DINT(_u.AlarmLog.Active[_slot].ResetClass),
        Message := 'AUTO_RESET, so it never blocks the commissioning it serves');
    AssertFalse(Condition := _u.AlarmLog.Blocking,
        Message := 'and Start stays available');
    // The whole point: no operator action closes this. OperatorReset reaches
    // only MANUAL_RESET events, and the rationalization record is not shelvable.
    _u.AlarmLog.OperatorReset();
    _u();
    AssertTrue(Condition := _u.AlarmLog.FindActiveSlot(SourcePath := 'Test.GateUnit',
        Description := 'std.engineering.simulation') > 0,
        Message := 'an operator reset does not clear it');
    AssertFalse(Condition := _u.AlarmLog.Shelve(Slot := _slot, DurationS := 60),
        Message := 'and shelving cannot silence it either');
    // It is raised ONCE per gate, however long the station runs.
    _u();
    _u();
    AssertEquals_INT(Expected := _gateMode.Count, Actual := _u.AlarmLog.NActive,
        Message := 'one standing event per REGISTERED gate, not one per scan');
    _w4 := TRUE;
END_IF
TEST_FINISHED();
END_METHOD

END_FUNCTION_BLOCK
